// TIA Portal V19 export
TYPE "Prod_Part_Area"
   STRUCT
      Halted { ExternalWritable := 'False'} : "Prod_Halted";
      Doors_Closed { ExternalWritable := 'False'} : Bool;
      Man { ExternalWritable := 'False'} : Bool;
      CycleON { ExternalWritable := 'False'} : Bool;
      Running { ExternalWritable := 'False'} : Bool;
      SetUpDone : Bool;
      SetupDone_Ax : Array[1..14] of Bool;
      MaterialPresenceEntry { ExternalWritable := 'False'} : Bool;
      MaterialPresenceExit { ExternalWritable := 'False'} : Bool;
      Material_Presence { ExternalWritable := 'False'} : Bool;
      MaterialFeedingStandstill { ExternalWritable := 'False'} : Bool;
      LeadCutMem { ExternalWritable := 'False'} : Bool;
      Material_Qty_FromLastCut { ExternalWritable := 'False'} : LReal;
   END_STRUCT;
END_TYPE
